ABB RobotStudio station: MultiTasking.rsstnx

Station MultiTasking (saved by RobotStudio 23.3.10550.0)
Controller IRB120FGL_3_58
  mechanical unit ROB_1: IRB120FGL_3_58__01, 6 joints, base frame (0, 0, 0) mm
Layout (positions relative to the parent item):
  - IRB120FGL_3_58__01 [mechanism, from %ABB.RobotStudio.Models.IRB120%\IRB120FGL_3_58__01.rslib] at (0, 0, 0) mm; joint values [0, 0, 0, 0, 0.5236, 0] (rad or m)
Targets, tools, work objects and paths stored in the station, written as RAPID:
! task T_ROB1
MODULE MainModule
  CONST robtarget Target_10:=[[-285.571688851,-254.029837254,381.276356624],[-0.000000084,-0.00000001,1,-0.000000053],[-2,-1,-2,0],[9E+09,9E+09,9E+09,9E+09,9E+09,9E+09]];
  CONST robtarget Target_20:=[[364.353829072,0,594],[0.5,0,0.866025404,0],[0,0,0,0],[9E+09,9E+09,9E+09,9E+09,9E+09,9E+09]];
  PROC Path_10()
    MoveL Target_10,v1000,z100,tool0\WObj:=wobj0;
    MoveJ Target_20,v1000,z100,tool0\WObj:=wobj0;
  ENDPROC
ENDMODULE

